// TIA Portal project "water" (V15)

(* hardware
DEVICE "HMI_1"  KTP700 Basic PN
   slot 0: "HMI_1"  KTP700 Basic PN  6AV2 123-2GB03-0AX0  15.0.0.0
   slot 1: "HMI_RT_1"  KTP700 Basic PN  6AV2 123-2GB03-0AX0  15.0.0.0
   slot 5: "HMI_1.IE_CP_1"  PROFINET Interface  15.0.0.0
      slot 1: "PROFINET Interface_1"  PROFINET Interface
         slot 1: "Port_1"  Port
DEVICE "S7300/ET200M station_1"  S7-300 station
   slot 0: "Rail_0"  Rail  6ES7 390-1***0-0AA0
   slot 2: "PLC_1"  CPU 314C-2 PN/DP  6ES7 314-6EH04-0AB0  V3.3
      slot 2: "PROFINET interface_1"  PN-IO
         slot 1: "Port_1"  Port
         slot 2: "Port_2"  Port
      slot 5: "DI 24/DO 16_1"  DI24/DO16
      slot 6: "AI 5/AO 2_1"  AI5/AO2
      slot 7: "Count_1"  Counter
      slot 8: "Positioning_1"  Positioning
*)

// ===== PLC "PLC_1"  CPU 314C-2 PN/DP =====

VAR_GLOBAL   // PLC tag table "Default tag table"
   "SP_INT" AT %MD4 : Real;
   "SENSOR" AT %IW30 : Word;
   "MAN_ON" AT %M0.0 : Bool;
   "PVPER_ON" AT %M0.1 : Bool;
   "LMN" AT %MD8 : Real;
   "P" AT %MD12 : Real;
   "I" AT %MD16 : Real;
   "D" AT %MD20 : Real;
   "PV" AT %MD24 : Real;
   "Tag_1" AT %MW28 : Word;
   "Tag_2" AT %QW30 : Word;
   "SEN" AT %ID30 : Real;
   "Tag_3" AT %QD30 : Real;
   "Tag_4" AT %MD50 : Real;
   "Tag_5" AT %MD30 : Real;
   "Tag_6" AT %QD34 : Real;
   "Tag_7" AT %QD32 : Real;
   "Tag_8" AT %MD60 : Real;
   "Tag_9" AT %MD65 : Real;
END_VAR

ORGANIZATION_BLOCK "Main"   // OB1, LAD
TITLE = "Main Program Sweep (Cycle)"
{ S7_Optimized_Access := 'FALSE' }
VERSION : 0.1
   VAR_TEMP
      OB1_EV_CLASS : Byte;   // Bits 0-3 = 1 (Coming event), Bits 4-7 = 1 (Event class 1)
      OB1_SCAN_1 : Byte;   // 1 (Cold restart scan 1 of OB 1), 3 (Scan 2-n of OB 1)
      OB1_PRIORITY : Byte;   // Priority of OB Execution
      OB1_OB_NUMBR : Byte;   // 1 (Organization block 1, OB1)
      OB1_RESERVED_1 : Byte;   // Reserved for system
      OB1_RESERVED_2 : Byte;   // Reserved for system
      OB1_PREV_CYCLE : Int;   // Cycle time of previous OB1 scan (milliseconds)
      OB1_MIN_CYCLE : Int;   // Minimum cycle time of OB1 (milliseconds)
      OB1_MAX_CYCLE : Int;   // Maximum cycle time of OB1 (milliseconds)
      OB1_DATE_TIME : Date_And_Time;   // Date and time OB1 started
   END_VAR
BEGIN

REGION Network 1
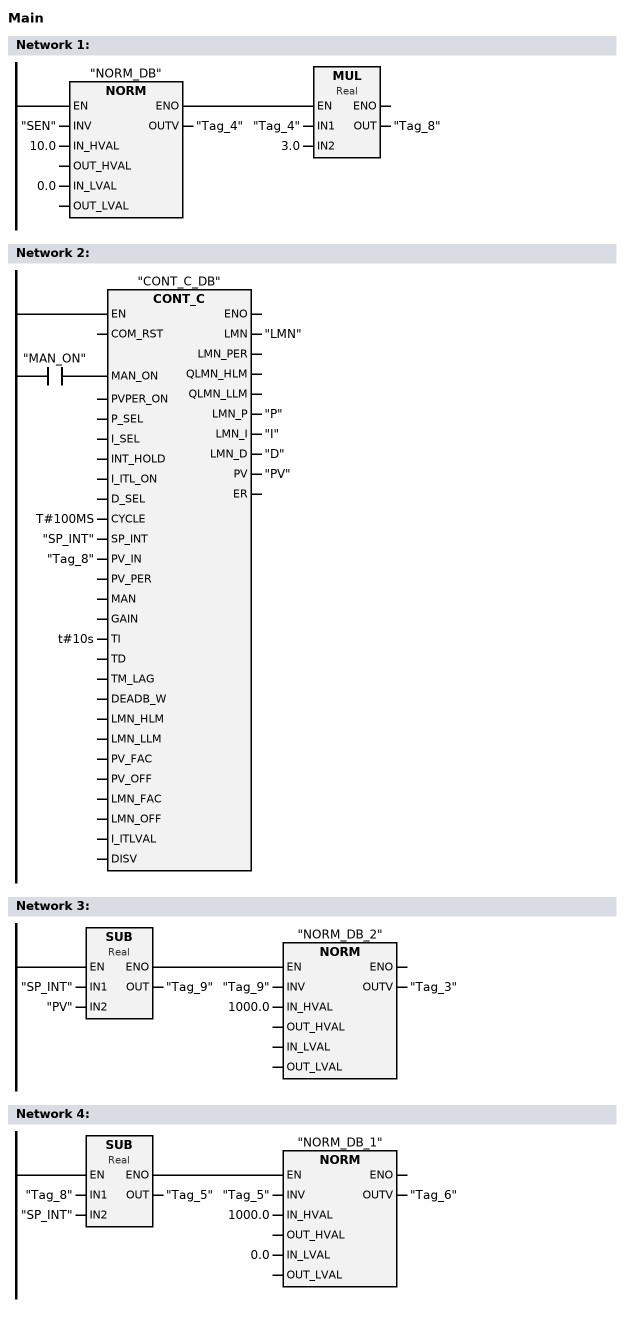
   // ENO of a box is taken as its EN; it also drops when the box reports an error
   "NORM_DB"(INV := "SEN", IN_HVAL := 10.0, IN_LVAL := 0.0, OUTV => "Tag_4");   // NORM
   "Tag_8" := "Tag_4" * 3.0;
END_REGION

REGION Network 2
   "CONT_C_DB"(MAN_ON := "MAN_ON",   // CONT_C
               CYCLE := T#100MS,
               SP_INT := "SP_INT",
               PV_IN := "Tag_8",
               TI := t#10s,
               LMN => "LMN",
               LMN_P => "P",
               LMN_I => "I",
               LMN_D => "D",
               PV => "PV");
END_REGION

REGION Network 3
   // ENO of a box is taken as its EN; it also drops when the box reports an error
   "Tag_9" := "SP_INT" - "PV";
   "NORM_DB_2"(INV := "Tag_9", IN_HVAL := 1000.0, OUTV => "Tag_3");   // NORM
END_REGION

REGION Network 4
   // ENO of a box is taken as its EN; it also drops when the box reports an error
   "Tag_5" := "Tag_8" - "SP_INT";
   "NORM_DB_1"(INV := "Tag_5", IN_HVAL := 1000.0, IN_LVAL := 0.0, OUTV => "Tag_6");   // NORM
END_REGION
END_ORGANIZATION_BLOCK

(* ===== HMI "HMI_RT_1" =====
system functions are stored by id; their names below are inferred from use
connection "HMI_Connection_1": ETHERNET, SIMATIC S7 300/400 MPI

HMI tags "Default tag table"
   "Tag_ScreenNumber" : UInt, internal
   "SP_INT" : Real = PLC SP_INT AT %MD4, 1 s
   "LMN" : Real = PLC LMN AT %MD8, 1 s
   "PV" : Real = PLC PV AT %MD24, 1 s
   "SENSOR" : Word = PLC SENSOR AT %IW30, 1 s
   "MAN_ON" : Bool = PLC MAN_ON AT %M0.0, 1 s
   "P" : Real = PLC P AT %MD12, 1 s
   "I" : Real = PLC I AT %MD16, 1 s
   "D" : Real = PLC D AT %MD20, 1 s
   "SEN" : Real = PLC SEN AT %ID30, 1 s
   "Tag_3" : Real = PLC Tag_3 AT %QD30, 1 s
   "Tag_5" : Real = PLC Tag_5 AT %MD30, 1 s
   "Tag_4" : Real = PLC Tag_4 AT %MD50, 1 s
   "Tag_9" : Real = PLC Tag_9 AT %MD65, 1 s

Template "Template_1" 800x480
   Button "Exit" at 714,429 size 71x50; TextOff 'Exit'; PictureOff "ExitRuntime_KTP700_Basic_PN_TR"; PictureOn "ExitRuntime_KTP700_Basic_PN_TR"
      on Release: StopRuntime(0)
   Button "Template_Button" at 614,429 size 71x50; TextOff 'Text'
   Button "Template_Button_1" at 514,429 size 71x50; TextOff 'Text'
   Button "Template_Button_2" at 414,429 size 71x50; TextOff 'Text'
   Button "Template_Button_3" at 314,429 size 71x50; TextOff 'Text'
   Button "Template_Button_4" at 214,429 size 71x50; TextOff 'Text'
   Button "Alarms" at 114,429 size 71x50; TextOff 'Alarms'; PictureOff "AlarmDisplay_KTP700_Basic_PN_TR"; PictureOn "AlarmDisplay_KTP700_Basic_PN_TR"
      on Release: function_ef3f5d25("Alarm window_Unacknowledged", -1)
   Button "Start screen" at 14,429 size 71x50; TextOff 'Start screen'; PictureOff "NavigateHome_KTP700_Basic_PN_TR"; PictureOn "NavigateHome_KTP700_Basic_PN_TR"
      on Release: ActivateScreen("Root screen", 0)
   SymbolicIOField "Symbolic_IO_Field_Screen" at 93,9 size 600x33; TextOff '0'; TextOn '1'; TextList "TextList_ScreenNames"
      ProcessValue <- "Tag_ScreenNumber"
      on Change: ActivateScreenByNumber("Tag_ScreenNumber", 0)
   DateTimeField "HmiScreenItemData" at 695,25 size 105x25
   DateTimeField "HmiScreenItemData_1" at 695,0 size 105x25
   GraphicView "Logo" at 0,0 size 91x51; Picture "Logo of HMI_1"

screen "Root screen" 800x480, template "Template_1"
   on GenerateScreen: SetTag("Tag_ScreenNumber", 1)
   TextField "HmiScreenItemData_2" at 80,225 size 640x25; Text 'Welcome to HMI_1 (KTP700 Basic+ PN)!'
   Button "HmiScreenItemData" at 36,87 size 159x47; TextOff 'LEVEL + SP'; TextOn 'SP + OP +PV'; PictureOff "Navigates to Screen0 for KTP700 Basic+ PN 15.0.0.0"; PictureOn "Navigates to Screen0 for KTP700 Basic+ PN 15.0.0.0"
      on Release: ActivateScreen("LEVEL + SP", 0)
   Button "HmiScreenItemData_1" at 36,146 size 159x47; TextOff 'PID'; PictureOff "Navigates to Screen1 for KTP700 Basic+ PN 15.0.0.0"; PictureOn "Navigates to Screen1 for KTP700 Basic+ PN 15.0.0.0"
      on Release: ActivateScreen("PID", 0)

screen "LEVEL + SP" 800x480, template "Template_1"
   on GenerateScreen: SetTag("Tag_ScreenNumber", 2)
   Button "Back" at 1,52 size 159x47; TextOff 'Back'
      on Release: ActivateScreen("Root screen", 0)
   TrendView "Trend view_1" at 1,101 size 600x324
   IOField "I/O field_1" at 614,99 size 96x32; FormatPattern s999999999.999
      ProcessValue <- "SP_INT"
   IOField "I/O field_4" at 614,162 size 96x32; FormatPattern s999999999.999
      ProcessValue <- "PV"
   Switch "Switch_1" at 286,58 size 110x32; CaptionText 'Switch'; TextOff 'AUTO'; TextOn 'MANUAL'
      ProcessValue <- "MAN_ON"
   TextField "Text field_1" at 614,68 size 26x23; Text 'SP'
   TextField "Text field_4" at 614,141 size 54x23; Text 'LEVEL'

screen "PID" 800x480, template "Template_1"
   on GenerateScreen: SetTag("Tag_ScreenNumber", 3)
   TextField "HmiScreenItemData" at 80,225 size 640x25; Text 'Screen1'
   Button "Back" at 1,52 size 159x47; TextOff 'Back'
      on Release: ActivateScreen("Root screen", 0)
   IOField "I/O field_1" at 614,99 size 96x32; FormatPattern s999999999.999
      ProcessValue <- "SP_INT"
   IOField "I/O field_3" at 614,164 size 96x32; FormatPattern s999999999.999
      ProcessValue <- "P"
   Switch "Switch_1" at 286,58 size 110x32; TextOn 'MANUAL'; CaptionText 'Switch'; TextOff 'AUTO'
      ProcessValue <- "MAN_ON"
   TextField "Text field_1" at 614,68 size 26x23; Text 'SP'
   TextField "Text field_3" at 613,141 size 16x23; Text 'P'
   TrendView "Trend view_1" at 1,101 size 600x324
   IOField "I/O field_4" at 614,238 size 96x32; FormatPattern s999999999.999
      ProcessValue <- "I"
   TextField "Text field_4" at 614,217 size 12x23; Text 'I'
   IOField "I/O field_5" at 614,307 size 96x32; FormatPattern s999999999.999
      ProcessValue <- "D"
   TextField "Text field_5" at 614,286 size 17x23; Text 'D'
*)